FUNCTION_BLOCK MetreCubeTime_Calculator (* Basic Function Block Type *)
  (* Standard: 61499-2 *)
  (* Version 0.0, 9/26/2024, SESA713705, Schneider Electric, Template *)
  PACKAGE SE.Nereda;
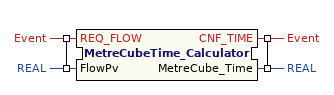
  EVENT_INPUT
    REQ_FLOW WITH FlowPv; (* Normal Execution Request *)
  END_EVENT
  EVENT_OUTPUT
    CNF_TIME WITH MetreCube_Time;
  END_EVENT
  VAR_INPUT
    FlowPv : REAL; (* Input event qualifier *)
  END_VAR
  VAR_OUTPUT
    MetreCube_Time : REAL;
  END_VAR
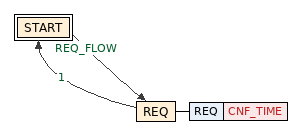
  EC_STATES
    START; (* Initial State *)
    REQ : REQ -> CNF_TIME; (* Normal execution *)
  END_STATES
  EC_TRANSITIONS
    START TO REQ := REQ_FLOW;
    REQ TO START := 1;
  END_TRANSITIONS
  ALGORITHM REQ IN ST: (* Normally executed algorithm *)
;
// We have time = V / Q; with V = Volume et Q = Flow; x3600 to convert it from Hour to s
IF FlowPv <> 0 AND FlowPv > 0.1 THEN
	MetreCube_Time := (1/ FlowPv) * 3600;
ELSE
	MetreCube_Time := 0;
END_IF;
  END_ALGORITHM
END_FUNCTION_BLOCK
